FUNCTION_BLOCK EL2808
VAR
	{attribute addProperty Name "WcState"}
	_wcState : WcStateBase;
	{attribute addProperty Name "Info data"}
	_infoData : InfoDataBase;
	_io : EL2xx8_Data;
END_VAR

PROPERTY IO : REFERENCE TO EL2xx8_Data
GET
IO REF= _io;
END_GET
END_PROPERTY

PROPERTY WcState : REFERENCE TO WcStateBase
GET
WcState REF= _wcState;
END_GET
END_PROPERTY

END_FUNCTION_BLOCK

(* stored: Version 1.1.0.1, ProductVersion 3.1.4024.9
   POU EL2808: Id {e7102656-8922-0390-341b-d82c51b6be4b}, SpecialFunc None
   Property IO: Id {affec52f-5d6c-0c2d-06de-86ac8b8272fa}
   Get Get: Id {0096a504-41b3-0c7f-2311-fd0d11133773}
   Property WcState: Id {75b368b6-6dd3-0c8e-1413-e5a756ab9f6b}
   Get Get: Id {c398bc87-ce28-033d-2c7c-19d6ea526d40} *)
